{attribute 'call_after_init'}
FUNCTION_BLOCK FB_FastFault_Test EXTENDS TcUnit.FB_TestSuite
VAR_INPUT
END_VAR
VAR_OUTPUT
END_VAR
VAR

END_VAR

FFCombinedFunctionality();
FFRegistration();

METHOD FFCombinedFunctionality
VAR_INPUT
END_VAR
VAR
	fbFF	:	FB_FastFault;
	fbFFO	:	FB_HardwareFFOutput;
	
END_VAR
TEST('FFCombinedFunctionality');

//Clear initial faults
fbFFO(i_xReset:=TRUE); //Reset requested at start of cycle

fbFF(io_fbFFHWO := fbFFO, //FF reset somehwere in code
	i_xOK := TRUE,
	i_xReset := TRUE);

fbFFO.EvaluateOutput(); //FFO eval called at end of cycle
	
AssertTrue(fbFFO.q_xFastFaultOut,
	'Fast fault did not clear');


//Induce fault with FF

fbFFO(i_xReset := FALSE); //Reset released at start of cycle

fbFF(io_fbFFHWO := fbFFO, //FF faulted
	i_xOK := FALSE); //Reset is still set true from last call.
	
fbFFO.EvaluateOutput(); //FFO eval called at end of cycle

AssertFalse(fbFFO.q_xFastFaultOut,
	'Fast fault did not trip the beam');
	
	
//FFO remains faulted until local (FF) and FFO receieve fresh reset request, and faults
//are actually cleared

//Attempt to clear FFO fails because FF still faulted
fbFFO(i_xReset := TRUE); //Reset requested

fbFF(io_fbFFHWO := fbFFO, //FF faulted
	i_xOK := FALSE,
	i_xReset := FALSE);
	
fbFFO.EvaluateOutput(); //FFO eval called at end of cycle

AssertFalse(fbFFO.q_xFastFaultOut,
	'Fast fault output cleared while fault remains, very bad');
	
//Attempt to clear FF while fault remains fails
fbFFO(i_xReset := FALSE);
fbFFO(i_xReset := TRUE); //Reset requested

fbFF(io_fbFFHWO := fbFFO, //FF faulted
	i_xOK := FALSE,
	i_xReset := TRUE); //This reset should fail.
	
fbFFO.EvaluateOutput(); //FFO eval called at end of cycle

AssertFalse(fbFFO.q_xFastFaultOut,
	'Fast fault cleared while fault remains, very bad');
	
TEST_FINISHED();
END_METHOD

METHOD FFRegistration
VAR_INPUT
END_VAR
VAR
	fbFF	:	FB_FastFault;
	fbFFO	:	FB_HardwareFFOutput;
END_VAR
TEST('FFRegistration');

fbFF(io_fbFFHWO := fbFFO);

AssertEquals_STRING(fbFF.sPath, fbFFO.asList[fbFFO.nIndex-1],
	'FF registration with FFO did not succeed');

TEST_FINISHED();
END_METHOD

END_FUNCTION_BLOCK

(* stored: Version 1.1.0.1, ProductVersion 3.1.4024.0
   POU FB_FastFault_Test: Id {c6666cf6-8125-0d8d-3cf9-a2348e99781e}, SpecialFunc None
   Method FFCombinedFunctionality: Id {40db6f61-8d2d-068a-122d-5b98f2f3d16e}
   Method FFRegistration: Id {d751f466-f83a-0e08-0ef0-631e8f42af98} *)
